FUNCTION F_softplus : lreal
VAR_INPUT
	x : LREAL;
END_VAR

IF x > 1E2 THEN
	F_softplus := x;
ELSIF x < -1E2 THEN
	F_softplus := 0;
ELSE
	F_softplus := LOG(EXP(x)+1);
END_IF

END_FUNCTION

(* stored: Version 1.1.0.1, ProductVersion 3.1.4024.12
   POU F_softplus: Id {595aca46-1dce-4de1-8177-d23da8043630}, SpecialFunc None *)
